(* CoDeSys 2.3 export: PLC_PRG.EXP *)

(* POU PLC_PRG, SFC *)
PROGRAM PLC_PRG
VAR
END_VAR
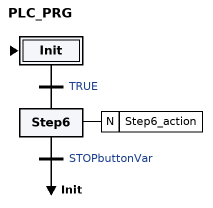
INITIAL_STEP Init:
END_STEP
TRANSITION FROM Init TO Step6 := TRUE;
END_TRANSITION
STEP Step6:
	Step6_action(N);
END_STEP
TRANSITION FROM Step6 TO Init := STOPbuttonVar;
END_TRANSITION

ACTION Step6_action:
PRG_MAIN;
Quel_Etage();
Priorite_Memo();
Appel_Palier();
Arret_Urgence();
ZAuto_RUN();
END_ACTION
END_PROGRAM
